// TwinCAT 3 PLC project Anker_Alserbachstrasse
// ProgramVersion: 3.1.4023.0
// libraries:
//   EfficientIO Communicator, * (EfficientIO)
//   Lynus Energy Basic, * (Lynus AG)
//   Lynus Persistent Data V1, * (Lynus AG)
//   Lynus Standards, * (Lynus AG)
//   Tc2_BABasic, * (Beckhoff Automation GmbH)
//   Tc2_Standard, * (Beckhoff Automation GmbH)
//   Tc2_System, * (Beckhoff Automation GmbH)
//   Tc2_Utilities, * (Beckhoff Automation GmbH)
//   Tc3_IotBase, * (Beckhoff Automation GmbH)
//   Tc3_JsonXml, * (Beckhoff Automation GmbH)
//   Tc3_Module, * (Beckhoff Automation GmbH)
// project tree:
//   / FastTask.TcTTO (not stored), MiddleTask.TcTTO, SlowTask.TcTTO (not stored)
//   FBs/ FB_Shelly_Pro1PM.TcPOU, FB_Shelly_Pro1PM_Helper.TcPOU (not stored), FB_TimeSwitch.TcPOU, FB_TimeSwitch_V2.TcPOU
//   POUs/ prg5529Con.TcPOU, prg5529EMS.TcPOU, prgComEffIO.TcPOU, prg5529Grid.TcPOU, prgPersistent.TcPOU, prgRWEffIO.TcPOU, prgVarEffIO.TcPOU (not stored), prg_SystemTime.TcPOU (not stored)
// real-time tasks:
//   TASK FastTask: cycle T#5ms, priority 19, ADS port 350
//   TASK MiddleTask: cycle T#10ms, priority 20, ADS port 351
//   TASK SlowTask: cycle T#20ms, priority 21, ADS port 352
// I/O:
//   DEVICE Device 1 (Beckhoff CCAT)
//   DEVICE Device 2 (CX-BK)
//     Box 1 (CX-BK)
// variable links:
//   Anker_Alserbachstrasse/Anker_Alserbachstrasse Instance <-> Device 2 (CX-BK)/Box 1 (CX-BK)
//     MiddleTask Inputs/prg5529Grid.fbGrid.fbKL3403.byStateCH1 <-> Term 3 (KL3403)/Channel 1/State
//     MiddleTask Inputs/prg5529Grid.fbGrid.fbKL3403.byStateCH2 <-> Term 3 (KL3403)/Channel 2/State
//     MiddleTask Inputs/prg5529Grid.fbGrid.fbKL3403.byStateCH3 <-> Term 3 (KL3403)/Channel 3/State
//     MiddleTask Inputs/prg5529Grid.fbGrid.fbKL3403.iDataInCH1 <-> Term 3 (KL3403)/Channel 1/Data In
//     MiddleTask Inputs/prg5529Grid.fbGrid.fbKL3403.iDataInCH2 <-> Term 3 (KL3403)/Channel 2/Data In
//     MiddleTask Inputs/prg5529Grid.fbGrid.fbKL3403.iDataInCH3 <-> Term 3 (KL3403)/Channel 3/Data In
//     MiddleTask Inputs/prg5529Grid.fbKBusState.uiKBusState_OUT <-> Inputs/State
//     MiddleTask Outputs/prg5529EMS.bQ1Switch <-> Term 2 (KL2408)/Channel 1/Output
//     MiddleTask Outputs/prg5529Grid.fbGrid.fbKL3403.byCntrCH1 <-> Term 3 (KL3403)/Channel 1/Ctrl
//     MiddleTask Outputs/prg5529Grid.fbGrid.fbKL3403.byCntrCH2 <-> Term 3 (KL3403)/Channel 2/Ctrl
//     MiddleTask Outputs/prg5529Grid.fbGrid.fbKL3403.byCntrCH3 <-> Term 3 (KL3403)/Channel 3/Ctrl

CONFIGURATION Anker_Alserbachstrasse
    RESOURCE PLC ON TwinCAT3
        TASK MiddleTask(INTERVAL := T#10ms, PRIORITY := 20);
        PROGRAM prg5529Grid WITH MiddleTask : prg5529Grid;
        PROGRAM prgPersistent WITH MiddleTask : prgPersistent;
        PROGRAM prg5529EMS WITH MiddleTask : prg5529EMS;
        PROGRAM prg5529Con WITH MiddleTask : prg5529Con;
    END_RESOURCE
END_CONFIGURATION

// ---- POUs/prg5529Grid.TcPOU
PROGRAM prg5529Grid
VAR
	fbKBusState		: FB_K_Bus_State;
	fbGrid			: FB_EM_Beckhoff_KL3403;
	lrPowerGrid		: LREAL;							//{#lynus.ag#()}
	lrCounterGrid	: LREAL;							//{#lynus.ag#()}
	lrVoltageGridL1	: LREAL;							//{#lynus.ag#()}
	lrVoltageGridL2	: LREAL;							//{#lynus.ag#()}
	lrVoltageGridL3	: LREAL;							//{#lynus.ag#()}
	uint_BusState	: UINT;								//{#lynus.ag#()}
END_VAR

//The mapping of this function must be linked with the K-Bus State in the E/A Part
fbKBusState(	uiKBusState_OUT=> , 
				b_Kbus_notOk=> , 
				word_ErrorCount=> );
				
//The mapping of this function must be linked with the KL3403 in the E/A Part
fbGrid(
	bEnable:= TRUE, 
	bChannel1Invers:= FALSE,					//Invert power data when transformer are mounted upside down
	bChannel2Invers:= FALSE,
	bChannel3Invers:= FALSE,
	uiCurrentTransformerRatioL1:= 400, 		//Transformer ratio on the secondary side
	uiCurrentTransformerRatioL2:= 400, 
	uiCurrentTransformerRatioL3:= 400, 
	uiKBusState_IN:= fbKBusState.uiKBusState_OUT, 
	stDataEMPower=> , 
	stDataEMCounter=> , 
	stDataEMPowerRealTime=> , 
	stDataEMCounterRealTime=> , 
	diNrOfEM_OUT=> );

lrPowerGrid := fbGrid.stDataEMPower.lrPowerTotal;
	lrCounterGrid := fbGrid.stDataEMCounter.lrTotalCounterEnergy_Consumption;	
		lrVoltageGridL1 := fbGrid.stDataEMPowerRealTime.lrVoltageL1N;
			lrVoltageGridL2 := fbGrid.stDataEMPowerRealTime.lrVoltageL2N;
				lrVoltageGridL3 := fbGrid.stDataEMPowerRealTime.lrVoltageL3N;

				
uint_BusState := fbKbusState.uiKBusState_OUT;

END_PROGRAM

// ---- POUs/prgPersistent.TcPOU
PROGRAM prgPersistent
VAR
	fbUSV		: FB_WritePersistentData_CX81xx;
END_VAR

fbUSV(
	eSaveModeData:= eUSVSaveMode.eSaveWhenPowerfail, 
	bLoadPersistentDataOk=> , 
	bPowerFailDetect=> , 
	bError=> , 
	bySaveProcess=> , 
	dwStorageLast24h=> , 
	udiErrorCode=> );
	
prg_SystemTime();

END_PROGRAM

// ---- POUs/prg5529EMS.TcPOU
PROGRAM prg5529EMS
VAR
	bQ1Switch	AT%Q*	: BOOL;						//{#lynus.ag#()}

	b_Coffee_Manual_On: BOOL;						//{#lynus.ag#()}
	b_Coffee_Manual_Off: BOOL;						//{#lynus.ag#()}
	b_AC_Manual_On: BOOL;							//{#lynus.ag#()}
	b_AC_Manual_Off: BOOL;							//{#lynus.ag#()}
	b_Vitrine_Manual_On: BOOL;						//{#lynus.ag#()}
	b_Vitrine_Manual_Off: BOOL;						//{#lynus.ag#()}
	b_Outside_Manual_On: BOOL;						//{#lynus.ag#()}
	b_Outside_Manual_Off: BOOL;						//{#lynus.ag#()}
	FB_TimeSwitch_Coffee: FB_TimeSwitch_V2;
//	FB_TimeSwitch_Coffee: FB_TimeSwitch;
	FB_TimeSwitch_AC: FB_TimeSwitch_V2;
//	FB_TimeSwitch_AC: FB_TimeSwitch;
	FB_TimeSwitch_Vitrine: FB_TimeSwitch_V2;
//	FB_TimeSwitch_Vitrine: FB_TimeSwitch;
	FB_TimeSwitch_Outside: FB_TimeSwitch_V2;
//	FB_TimeSwitch_Outside: FB_TimeSwitch;
	fbCalcSunriseSunset   		: FB_CalcSunriseSunset;
	todSunrise            		: TOD;
	todSunset             		: TOD;
	fb_GetTimeZoneInfo	:FB_GetTimeZoneInformation;
	b_firstCycle: BOOL;
	RS_Outsidelight: RS;
	r_trig_on: R_trig;
	r_trig_off: R_trig;
	b_Status_CoffeeMaschine: BOOL;					//{#lynus.ag#()}
	// not used any more
	m_error_test	:BOOL;								//{#lynus.ag#()}

END_VAR
VAR PERSISTENT
// opening hours	
	byte_MoFr_Open_Hour		:BYTE;								//{#lynus.ag#()}
	byte_MoFr_Open_Minute	:BYTE;								//{#lynus.ag#()}
	byte_MoFr_Close_Hour	:BYTE;								//{#lynus.ag#()}
	byte_MoFr_Close_Minute	:BYTE;								//{#lynus.ag#()}
	byte_Sa_Open_Hour		:BYTE;								//{#lynus.ag#()}
	byte_Sa_Open_Minute		:BYTE;								//{#lynus.ag#()}
	byte_Sa_Close_Hour		:BYTE;								//{#lynus.ag#()}
	byte_Sa_Close_Minute	:BYTE;								//{#lynus.ag#()}
	byte_So_Open_Hour		:BYTE;								//{#lynus.ag#()}
	byte_So_Open_Minute		:BYTE;								//{#lynus.ag#()}
	byte_So_Close_Hour		:BYTE;								//{#lynus.ag#()}
	byte_So_Close_Minute	:BYTE;								//{#lynus.ag#()}
	
// offset coffeemaschine in hours			
	b_Enable_Control_Coffee		:BOOL;								//{#lynus.ag#()}
	real_Coffee_Offset_Start	:REAL;								//{#lynus.ag#()}
	real_Coffee_Offset_Stop		:REAL;								//{#lynus.ag#()}

// offset AC in hours			
	b_Enable_Control_AC			:BOOL;								//{#lynus.ag#()}
	real_AC_Offset_Start		:REAL;								//{#lynus.ag#()}
	real_AC_Offset_Stop			:REAL;								//{#lynus.ag#()}
	
// offset Vitrine Cooler in hours			
	b_Enable_Control_Vitrine	:BOOL;								//{#lynus.ag#()}
	real_Vitrine_Offset_Start	:REAL;								//{#lynus.ag#()}
	real_Vitrine_Offset_Stop	:REAL;								//{#lynus.ag#()}

// offset outside light in hours			
	b_Enable_Control_Outside	:BOOL;								//{#lynus.ag#()}
	real_Outside_Offset_Start	:REAL;								//{#lynus.ag#()}
	real_Outside_Offset_Stop	:REAL;								//{#lynus.ag#()}
END_VAR

FB_TimeSwitch_Coffee(
	b_Enable:= b_Enable_Control_Coffee, 
	b_StatusOn:= NOT bQ1Switch, 
	structSystemTime:= prg_SystemTime.structSystemTime, 
	byte_MoFr_Open_Hour:= byte_MoFr_Open_Hour , 
	byte_MoFr_Open_Minute:= byte_MoFr_Open_Minute, 
	byte_MoFr_Close_Hour:= byte_MoFr_Close_Hour , 
	byte_MoFr_Close_Minute:= byte_MoFr_Close_Minute, 
	byte_Sa_Open_Hour:= byte_Sa_Open_Hour, 
	byte_Sa_Open_Minute:= byte_Sa_Open_Minute , 
	byte_Sa_Close_Hour:= byte_Sa_Close_Hour , 
	byte_Sa_Close_Minute:= byte_Sa_Close_Minute, 
	byte_So_Open_Hour:= byte_So_Open_Hour, 
	byte_So_Open_Minute:= byte_So_Open_Minute, 
	byte_So_Close_Hour:= byte_So_Close_Hour, 
	byte_So_Close_Minute:= byte_So_Close_Minute, 
	real_Offset_Start:= real_Coffee_Offset_Start , 
	real_Offset_Stop:= real_Coffee_Offset_Stop , 
	b_On_Manual:= b_Coffee_Manual_On, 
	b_Off_Manual:= b_Coffee_Manual_Off, 
	b_Output_On=> , 
	b_Error=> );
	
IF NOT FB_TimeSwitch_Coffee.b_Output_On THEN
	bQ1Switch := TRUE;
ELSIF FB_TimeSwitch_Coffee.b_Output_On THEN
	bQ1Switch := FALSE;
END_IF	
b_Status_CoffeeMaschine := NOT bQ1Switch;
	
FB_TimeSwitch_AC(
	b_Enable:= b_Enable_Control_AC, 
	b_StatusOn:=  prg5529CON.fbShelly[1].bStateP1, 
	structSystemTime:= prg_SystemTime.structSystemTime , 
	byte_MoFr_Open_Hour:= byte_MoFr_Open_Hour , 
	byte_MoFr_Open_Minute:= byte_MoFr_Open_Minute, 
	byte_MoFr_Close_Hour:= byte_MoFr_Close_Hour , 
	byte_MoFr_Close_Minute:= byte_MoFr_Close_Minute, 
	byte_Sa_Open_Hour:= byte_Sa_Open_Hour, 
	byte_Sa_Open_Minute:= byte_Sa_Open_Minute , 
	byte_Sa_Close_Hour:= byte_Sa_Close_Hour , 
	byte_Sa_Close_Minute:= byte_Sa_Close_Minute, 
	byte_So_Open_Hour:= byte_So_Open_Hour, 
	byte_So_Open_Minute:= byte_So_Open_Minute, 
	byte_So_Close_Hour:= byte_So_Close_Hour, 
	byte_So_Close_Minute:= byte_So_Close_Minute, 
	real_Offset_Start:= real_AC_Offset_Start , 
	real_Offset_Stop:= real_AC_Offset_Stop , 
	b_On_Manual:= b_AC_Manual_On, 
	b_Off_Manual:= b_AC_Manual_Off, 
	b_Output_On=> , 
	b_Error=> );

FB_TimeSwitch_Vitrine(
	b_Enable:= b_Enable_Control_Vitrine, 
	b_StatusOn:=  prg5529CON.fbShelly[3].bStateP1, 
	structSystemTime:= prg_SystemTime.structSystemTime , 
	byte_MoFr_Open_Hour:= byte_MoFr_Open_Hour , 
	byte_MoFr_Open_Minute:= byte_MoFr_Open_Minute, 
	byte_MoFr_Close_Hour:= byte_MoFr_Close_Hour , 
	byte_MoFr_Close_Minute:= byte_MoFr_Close_Minute, 
	byte_Sa_Open_Hour:= byte_Sa_Open_Hour, 
	byte_Sa_Open_Minute:= byte_Sa_Open_Minute , 
	byte_Sa_Close_Hour:= byte_Sa_Close_Hour , 
	byte_Sa_Close_Minute:= byte_Sa_Close_Minute, 
	byte_So_Open_Hour:= byte_So_Open_Hour, 
	byte_So_Open_Minute:= byte_So_Open_Minute, 
	byte_So_Close_Hour:= byte_So_Close_Hour, 
	byte_So_Close_Minute:= byte_So_Close_Minute, 
	real_Offset_Start:= real_Vitrine_Offset_Start , 
	real_Offset_Stop:= real_Vitrine_Offset_Stop , 
	b_On_Manual:= b_Vitrine_Manual_On, 
	b_Off_Manual:= b_Vitrine_Manual_Off, 
	b_Output_On=> , 
	b_Error=> );

// Sehlly 5 Outside light
FB_TimeSwitch_Outside(		
	b_Enable:= b_Enable_Control_Outside, 
	b_StatusOn:=  prg5529CON.fbShelly[5].bStateP1 , 
	structSystemTime:= prg_SystemTime.structSystemTime , 
	byte_MoFr_Open_Hour:= byte_MoFr_Open_Hour , 
	byte_MoFr_Open_Minute:= byte_MoFr_Open_Minute, 
	byte_MoFr_Close_Hour:= byte_MoFr_Close_Hour , 
	byte_MoFr_Close_Minute:= byte_MoFr_Close_Minute, 
	byte_Sa_Open_Hour:= byte_Sa_Open_Hour, 
	byte_Sa_Open_Minute:= byte_Sa_Open_Minute , 
	byte_Sa_Close_Hour:= byte_Sa_Close_Hour , 
	byte_Sa_Close_Minute:= byte_Sa_Close_Minute, 
	byte_So_Open_Hour:= byte_So_Open_Hour, 
	byte_So_Open_Minute:= byte_So_Open_Minute, 
	byte_So_Close_Hour:= byte_So_Close_Hour, 
	byte_So_Close_Minute:= byte_So_Close_Minute, 
	real_Offset_Start:= real_Outside_Offset_Start , 
	real_Offset_Stop:= real_Outside_Offset_Stop , 
	b_On_Manual:= b_Outside_Manual_On, 
	b_Off_Manual:= b_Outside_Manual_Off, 
	b_Output_On=> , 
	b_Error=> );
	
// calculate sunset / sunrise
// find out the time details
fb_GetTimeZoneInfo(
	sNetID:= '', 
	bExecute:= prg_SystemTime.structSystemTime.wHour = 4 OR NOT b_firstCycle, 
	tTimeout:= T#5S, 
	bBusy=> , 
	bError=> , 
	nErrID=> , 
	tzID=> , 
	tzInfo=> );
b_firstCycle := TRUE;

fbCalcSunriseSunset(
	fDegreeOfLongitude := 16.3731,   (* Longitude of Vienna *)
	fDegreeOfLatitude := 48.2083,   (* Latitude of Vienna*)
	fReferenceMeridian := SEL( fb_GetTimeZoneInfo.tzID = eTimeZoneID_Daylight ,15,30),  (* Central European Time 15 Winter Timer / 30 Summer Time *)
	dCurrentDate := DT_TO_DATE(SYSTEMTIME_TO_Dt (prg_SystemTime.structSystemTime)),
	todSunrise => todSunrise,
	todSunset => todSunset);
	
r_trig_on (clk := FB_TimeSwitch_Outside.b_Output_On AND DT_TO_TOD(systemtime_to_dt(prg_SystemTime.structSystemTime))< (todSunrise +  T#1H) );
r_trig_off (clk := NOT FB_TimeSwitch_Outside.b_Output_On);

RS_Outsidelight(	Set := r_trig_on.Q OR ((todSunset - T#2H) =  DT_TO_TOD(systemtime_to_dt(prg_SystemTime.structSystemTime)) AND FB_TimeSwitch_Outside.b_Output_On) OR b_Outside_Manual_On ,
					Reset1 := r_trig_off.Q OR ((todSunrise +  T#1H)= DT_TO_TOD(systemtime_to_dt(prg_SystemTime.structSystemTime))) OR b_Outside_Manual_Off,
					Q1 => );

END_PROGRAM

// ---- FBs/FB_TimeSwitch_V2.TcPOU
FUNCTION_BLOCK FB_TimeSwitch_V2
VAR_INPUT
	b_Enable: BOOL;
	b_StatusOn: BOOL;
	structSystemTime: timestruct;
	byte_MoFr_Open_Hour: BYTE;
	byte_MoFr_Open_Minute: BYTE;
	byte_MoFr_Close_Hour: BYTE;
	byte_MoFr_Close_Minute: BYTE;
	byte_Sa_Open_Hour: BYTE;
	byte_Sa_Open_Minute: BYTE;
	byte_Sa_Close_Hour: BYTE;
	byte_Sa_Close_Minute: BYTE;	
	byte_So_Open_Hour: BYTE;
	byte_So_Open_Minute: BYTE;
	byte_So_Close_Hour: BYTE;
	byte_So_Close_Minute: BYTE;
	real_Offset_Start: REAL;
	real_Offset_Stop: REAL;	
	b_On_Manual: BOOL;
	b_Off_Manual: BOOL;
END_VAR
VAR_OUTPUT
	b_Output_On: BOOL;
	b_Error: BOOL;
END_VAR
VAR
	TON_0: ton;
	byte_Day :BYTE;		// 0: Sunday, 1: Monday,....
	time_now             		: TIME;
	time_MoFr_Open             	: TIME;
	time_MoFr_Close             : TIME;
	time_Sa_Open             	: TIME;
	time_Sa_Close             	: TIME;
	time_So_Open             	: TIME;
	time_So_Close             	: TIME;
	

	RS_0: rs;
	R_TRIG_0: r_trig;
	R_TRIG_1: r_trig;
	dt_Test: DATE_AND_TIME;
	tod_test: TIME_OF_DAY;
	time_temp: TIME;
	time_Start_MoFr_Calc: TIME;
	time_Stop_MoFr_Calc: TIME;
	time_Start_Sa_Calc: TIME;
	time_Stop_Sa_Calc: TIME;
	time_Start_So_Calc: TIME;
	time_Stop_So_Calc: TIME;
	
	FB_WeeklyTimeSwitch_MoFr: FB_WeeklyTimeSwitch;
	FB_WeeklyTimeSwitch_Sa: FB_WeeklyTimeSwitch;
	FB_WeeklyTimeSwitch_So: FB_WeeklyTimeSwitch;
	RS_manu: rs;
	b_Auto_on: BOOL;

	R_TRIG_2: r_trig;
	R_TRIG_3: r_trig;
	F_TRIG_0: f_trig;
	R_TRIG_4: r_trig;
	R_TRIG_FirstCycle: r_trig;
	time_Zero             	: TIME;
	
END_VAR
VAR // added by the converter: edge detectors and wires of the graphical bodies
    _w1 : DATE_AND_TIME;
    _w2 : TIME_OF_DAY;
    _w3 : BOOL;
END_VAR

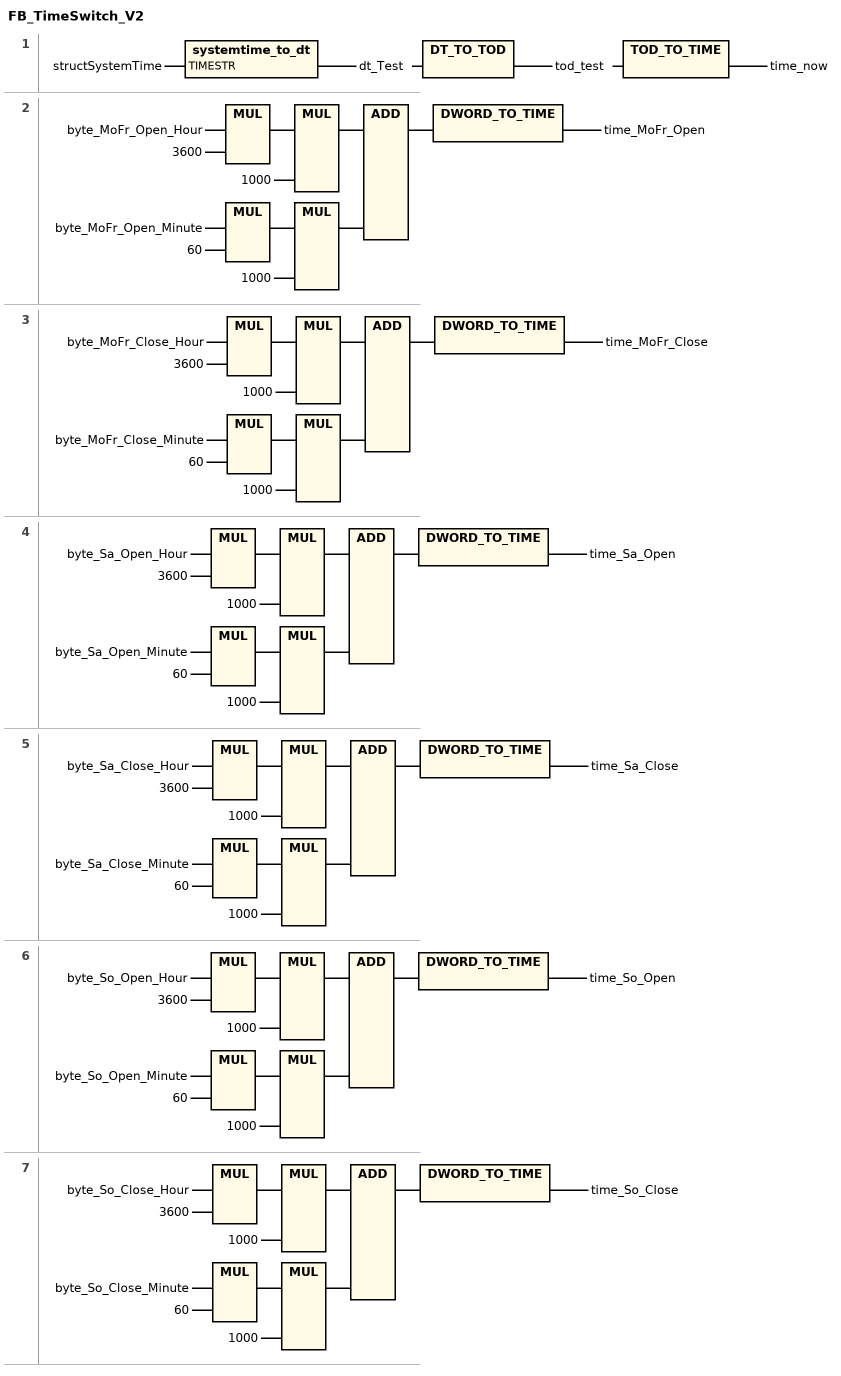
// NETWORK 1
_w1 := systemtime_to_dt(TIMESTR := structSystemTime);
dt_Test := _w1;
_w2 := DT_TO_TOD(_w1);
tod_test := _w2;
time_now := TOD_TO_TIME(_w2);

// NETWORK 2
time_MoFr_Open := DWORD_TO_TIME((byte_MoFr_Open_Hour * 3600) * 1000 + (byte_MoFr_Open_Minute * 60) * 1000);

// NETWORK 3
time_MoFr_Close := DWORD_TO_TIME((byte_MoFr_Close_Hour * 3600) * 1000 + (byte_MoFr_Close_Minute * 60) * 1000);

// NETWORK 4
time_Sa_Open := DWORD_TO_TIME((byte_Sa_Open_Hour * 3600) * 1000 + (byte_Sa_Open_Minute * 60) * 1000);

// NETWORK 5
time_Sa_Close := DWORD_TO_TIME((byte_Sa_Close_Hour * 3600) * 1000 + (byte_Sa_Close_Minute * 60) * 1000);

// NETWORK 6
time_So_Open := DWORD_TO_TIME((byte_So_Open_Hour * 3600) * 1000 + (byte_So_Open_Minute * 60) * 1000);

// NETWORK 7
time_So_Close := DWORD_TO_TIME((byte_So_Close_Hour * 3600) * 1000 + (byte_So_Close_Minute * 60) * 1000);

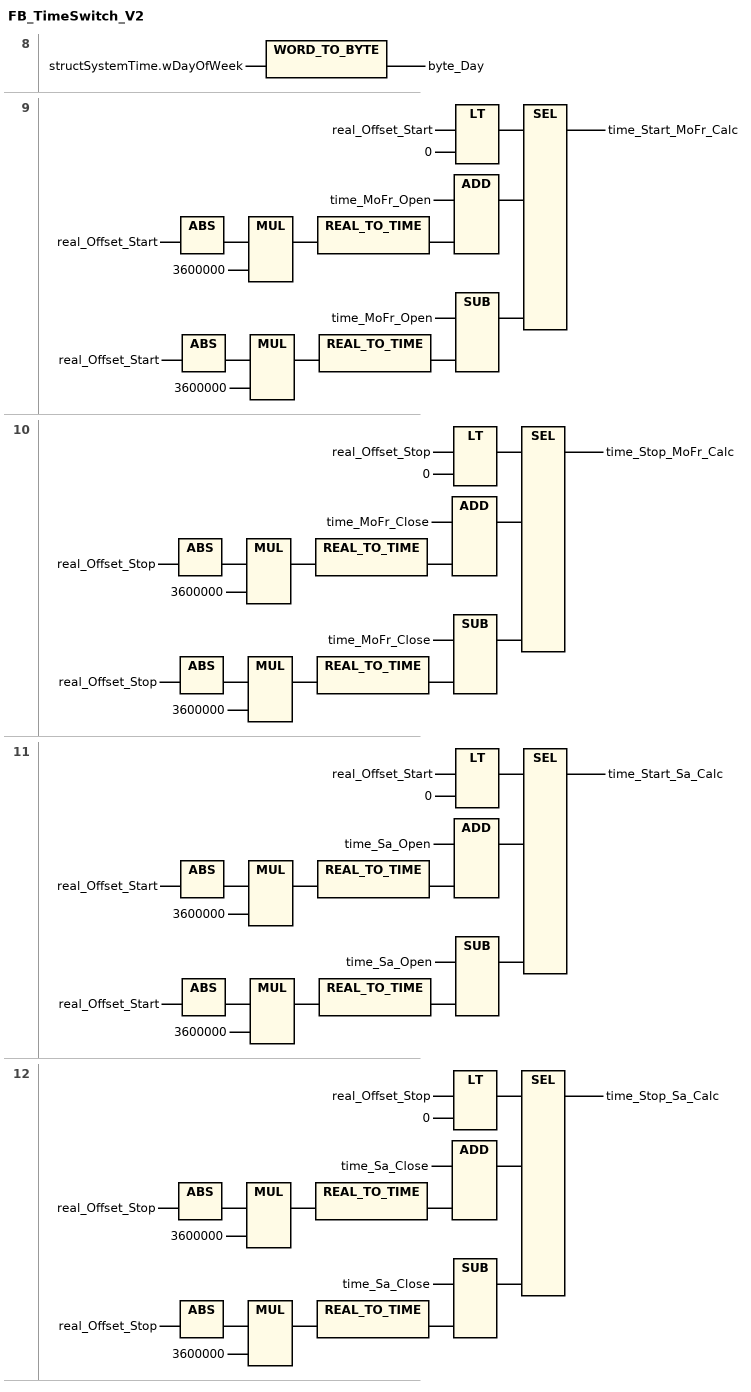
// NETWORK 8
byte_Day := WORD_TO_BYTE(structSystemTime.wDayOfWeek);

// NETWORK 9
time_Start_MoFr_Calc := SEL(real_Offset_Start < 0, time_MoFr_Open + REAL_TO_TIME(ABS(real_Offset_Start) * 3600000), time_MoFr_Open - REAL_TO_TIME(ABS(real_Offset_Start) * 3600000));

// NETWORK 10
time_Stop_MoFr_Calc := SEL(real_Offset_Stop < 0, time_MoFr_Close + REAL_TO_TIME(ABS(real_Offset_Stop) * 3600000), time_MoFr_Close - REAL_TO_TIME(ABS(real_Offset_Stop) * 3600000));

// NETWORK 11
time_Start_Sa_Calc := SEL(real_Offset_Start < 0, time_Sa_Open + REAL_TO_TIME(ABS(real_Offset_Start) * 3600000), time_Sa_Open - REAL_TO_TIME(ABS(real_Offset_Start) * 3600000));

// NETWORK 12
time_Stop_Sa_Calc := SEL(real_Offset_Stop < 0, time_Sa_Close + REAL_TO_TIME(ABS(real_Offset_Stop) * 3600000), time_Sa_Close - REAL_TO_TIME(ABS(real_Offset_Stop) * 3600000));

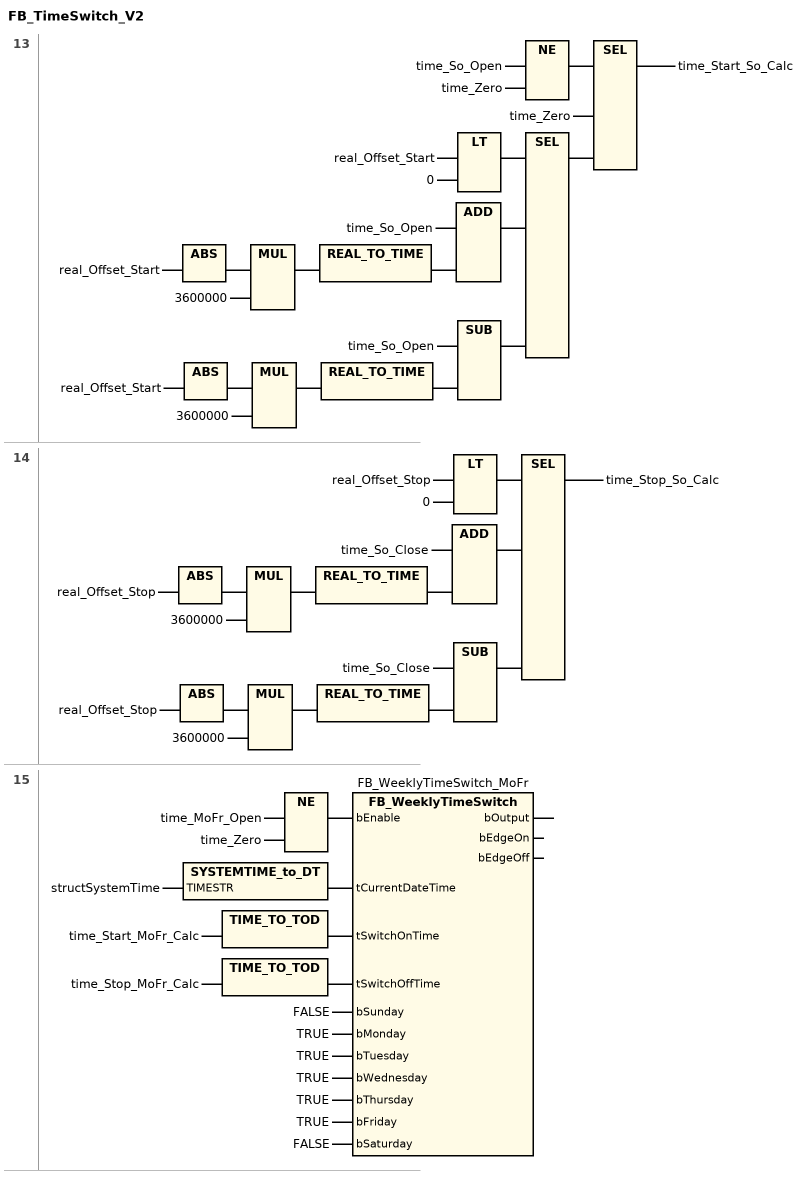
// NETWORK 13
time_Start_So_Calc := SEL(time_So_Open <> time_Zero, time_Zero, SEL(real_Offset_Start < 0, time_So_Open + REAL_TO_TIME(ABS(real_Offset_Start) * 3600000), time_So_Open - REAL_TO_TIME(ABS(real_Offset_Start) * 3600000)));

// NETWORK 14
time_Stop_So_Calc := SEL(real_Offset_Stop < 0, time_So_Close + REAL_TO_TIME(ABS(real_Offset_Stop) * 3600000), time_So_Close - REAL_TO_TIME(ABS(real_Offset_Stop) * 3600000));

// NETWORK 15
FB_WeeklyTimeSwitch_MoFr(
    bEnable := time_MoFr_Open <> time_Zero,
    tCurrentDateTime := SYSTEMTIME_to_DT(TIMESTR := structSystemTime),
    tSwitchOnTime := TIME_TO_TOD(time_Start_MoFr_Calc),
    tSwitchOffTime := TIME_TO_TOD(time_Stop_MoFr_Calc),
    bSunday := FALSE,
    bMonday := TRUE,
    bTuesday := TRUE,
    bWednesday := TRUE,
    bThursday := TRUE,
    bFriday := TRUE,
    bSaturday := FALSE); // FB_WeeklyTimeSwitch

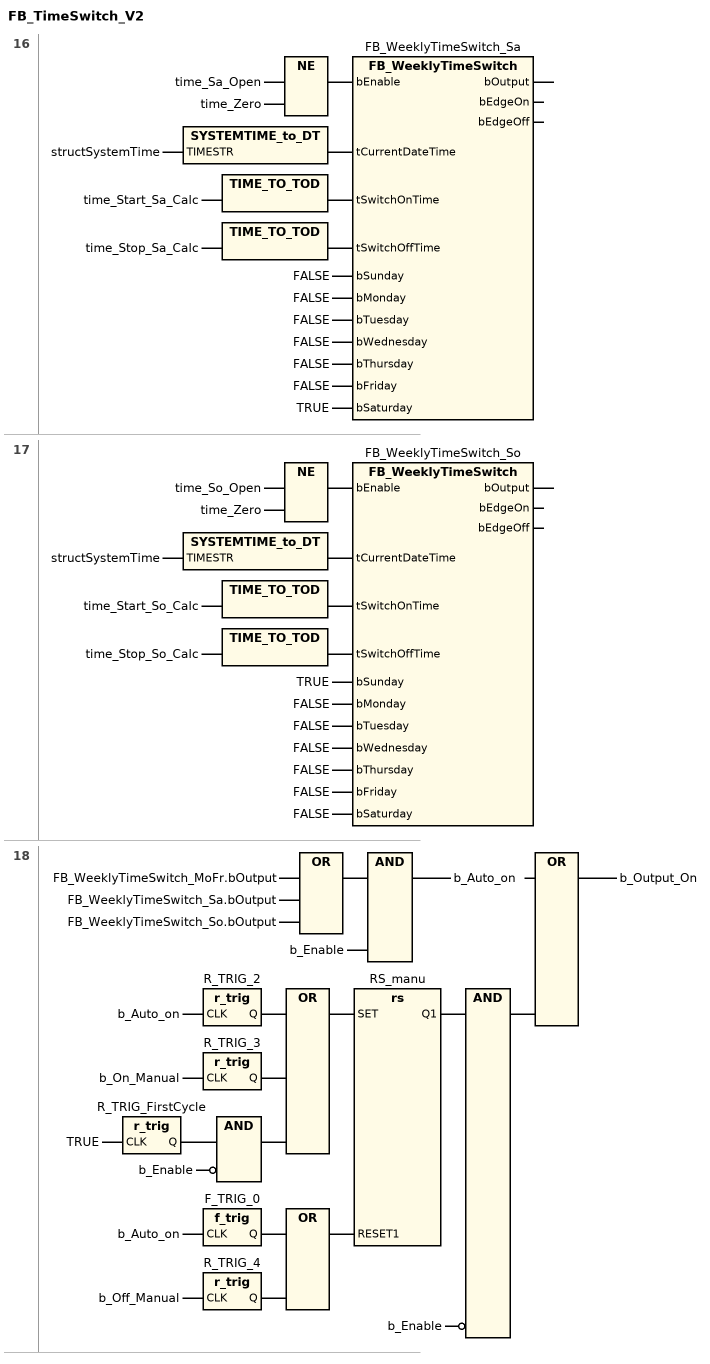
// NETWORK 16
FB_WeeklyTimeSwitch_Sa(
    bEnable := time_Sa_Open <> time_Zero,
    tCurrentDateTime := SYSTEMTIME_to_DT(TIMESTR := structSystemTime),
    tSwitchOnTime := TIME_TO_TOD(time_Start_Sa_Calc),
    tSwitchOffTime := TIME_TO_TOD(time_Stop_Sa_Calc),
    bSunday := FALSE,
    bMonday := FALSE,
    bTuesday := FALSE,
    bWednesday := FALSE,
    bThursday := FALSE,
    bFriday := FALSE,
    bSaturday := TRUE); // FB_WeeklyTimeSwitch

// NETWORK 17
FB_WeeklyTimeSwitch_So(
    bEnable := time_So_Open <> time_Zero,
    tCurrentDateTime := SYSTEMTIME_to_DT(TIMESTR := structSystemTime),
    tSwitchOnTime := TIME_TO_TOD(time_Start_So_Calc),
    tSwitchOffTime := TIME_TO_TOD(time_Stop_So_Calc),
    bSunday := TRUE,
    bMonday := FALSE,
    bTuesday := FALSE,
    bWednesday := FALSE,
    bThursday := FALSE,
    bFriday := FALSE,
    bSaturday := FALSE); // FB_WeeklyTimeSwitch

// NETWORK 18
_w3 := (FB_WeeklyTimeSwitch_MoFr.bOutput OR FB_WeeklyTimeSwitch_Sa.bOutput OR FB_WeeklyTimeSwitch_So.bOutput) AND b_Enable;
b_Auto_on := _w3;
R_TRIG_2(CLK := b_Auto_on); // r_trig
R_TRIG_3(CLK := b_On_Manual); // r_trig
R_TRIG_FirstCycle(CLK := TRUE); // r_trig
F_TRIG_0(CLK := b_Auto_on); // f_trig
R_TRIG_4(CLK := b_Off_Manual); // r_trig
RS_manu(SET := R_TRIG_2.Q OR R_TRIG_3.Q OR R_TRIG_FirstCycle.Q AND NOT b_Enable, RESET1 := F_TRIG_0.Q OR R_TRIG_4.Q); // rs
b_Output_On := _w3 OR RS_manu.Q1 AND NOT b_Enable;

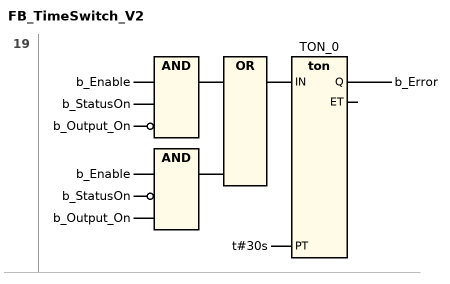
// NETWORK 19
TON_0(IN := b_Enable AND b_StatusOn AND NOT b_Output_On OR b_Enable AND NOT b_StatusOn AND b_Output_On, PT := t#30s); // ton
b_Error := TON_0.Q;

END_FUNCTION_BLOCK

// ---- POUs/prg5529Con.TcPOU
PROGRAM prg5529Con
VAR

	fbShelly				:	ARRAY[1..20] OF FB_Shelly_Pro1PM;
	f_Trig_Busy				:	ARRAY[1..20] OF f_trig;
			
//	fbShelly1				:	FB_Shelly_Pro1PM;
	lrS1P1Power				:	LREAL;			//{#lynus.ag#()}
	lrS1P1Power_kW			:	LREAL;			//{#lynus.ag#()}
	lrS1P1Voltage			:	LREAL;			//{#lynus.ag#()}
	lrS1P1Energy			:	LREAL;			//{#lynus.ag#()}
	lrS1P1Temperature		:	LREAL;			//{#lynus.ag#()}
	bS1P1On					:	BOOL;			//{#lynus.ag#()}
	bS1P1Off				:	BOOL;			//{#lynus.ag#()}
	bS1P1Switch				:	BOOL;			//{#lynus.ag#()}
	
	// Shelly2: 
//	fbShelly2				:	FB_Shelly_Pro1PM;
	lrS2P1Power				:	LREAL;			//{#lynus.ag#()}
	lrS2P1Power_kW			:	LREAL;			//{#lynus.ag#()}
	lrS2P1Voltage			:	LREAL;			//{#lynus.ag#()}
	lrS2P1Energy			:	LREAL;			//{#lynus.ag#()}
	lrS2P1Temperature		:	LREAL;			//{#lynus.ag#()}
	bS2P1On					:	BOOL;			//{#lynus.ag#()}
	bS2P1Off				:	BOOL;			//{#lynus.ag#()}
	bS2P1Switch				:	BOOL;			//{#lynus.ag#()}
	
	// Shelly3: 
//	fbShelly3				:	FB_Shelly_Pro1PM;
	lrS3P1Power				:	LREAL;			//{#lynus.ag#()}
	lrS3P1Power_kW			:	LREAL;			//{#lynus.ag#()}
	lrS3P1Voltage			:	LREAL;			//{#lynus.ag#()}
	lrS3P1Energy			:	LREAL;			//{#lynus.ag#()}
	lrS3P1Temperature		:	LREAL;			//{#lynus.ag#()}
	bS3P1On					:	BOOL;			//{#lynus.ag#()}
	bS3P1Off				:	BOOL;			//{#lynus.ag#()}
	bS3P1Switch				:	BOOL;			//{#lynus.ag#()}
	
	// Shelly4: 
//	fbShelly4				:	FB_Shelly_Pro1PM;
	lrS4P1Power				:	LREAL;			//{#lynus.ag#()}
	lrS4P1Power_kW			:	LREAL;			//{#lynus.ag#()}
	lrS4P1Voltage			:	LREAL;			//{#lynus.ag#()}
	lrS4P1Energy			:	LREAL;			//{#lynus.ag#()}
	lrS4P1Temperature		:	LREAL;			//{#lynus.ag#()}
	bS4P1On					:	BOOL;			//{#lynus.ag#()}
	bS4P1Off				:	BOOL;			//{#lynus.ag#()}
	bS4P1Switch				:	BOOL;			//{#lynus.ag#()}
	
	// Shelly5: 
//	fbShelly5				:	FB_Shelly_Pro1PM;
	lrS5P1Power				:	LREAL;			//{#lynus.ag#()}
	lrS5P1Power_kW			:	LREAL;			//{#lynus.ag#()}
	lrS5P1Voltage			:	LREAL;			//{#lynus.ag#()}
	lrS5P1Energy			:	LREAL;			//{#lynus.ag#()}
	lrS5P1Temperature		:	LREAL;			//{#lynus.ag#()}
	bS5P1On					:	BOOL;			//{#lynus.ag#()}
	bS5P1Off				:	BOOL;			//{#lynus.ag#()}
	bS5P1Switch				:	BOOL;			//{#lynus.ag#()}
	

	// Other
	lrRemainPower_kW		:	LREAL;			//{#lynus.ag#()}
	
	// state maschine for GET requests
	str_Array_IPs			: array[1..30] of STRING(15);			//arrays for IPs
	int_State: INT;													// state
	// Shelly: 


	int_Multiplier_1 			:INT:=1;								// multilpier received values, =2 when external fuse is on, was at the beginning
	int_Multiplier_2 			:INT:=2;								// multilpier received values, =2 when external fuse is on, was at the beginning
	int_Multiplier_3 			:INT:=1;								// multilpier received values, =2 when external fuse is on, was at the beginning
	int_Multiplier_4 			:INT:=2;								// multilpier received values, =2 when external fuse is on, was at the beginning
	int_Multiplier_5 			:INT:=1;								// multilpier received values, =2 when external fuse is on, was at the beginning
	int_TimeoutCounter: ARRAY[1..30] OF INT;	
	int_SuccessCounter: ARRAY[1..30] OF INT;	
	int_ErrorCounter: ARRAY[1..30] OF INT;
	ton_wait: Ton;
	mTest: BOOL;
	m_Error_HTTP: BOOL;							//{#lynus.ag#()}
END_VAR


CASE int_State OF
	0: 		// Init State
	
	// define IPs
	str_Array_IPs[1]	:='10.55.29.131';
	str_Array_IPs[2]	:='10.55.29.132';
	str_Array_IPs[3]	:='10.55.29.133';
	str_Array_IPs[4]	:='10.55.29.134';
	str_Array_IPs[5]	:='10.55.29.135';
	str_Array_IPs[6]	:='';
	str_Array_IPs[7]	:='';
	str_Array_IPs[8]	:='';
	str_Array_IPs[9]	:='';
	str_Array_IPs[10]	:='';
	str_Array_IPs[11]	:='';
	str_Array_IPs[12]	:='';
	str_Array_IPs[13]	:='';
	str_Array_IPs[14]	:='';
	fbShelly[1].sHostname:= str_Array_IPs[1];
	fbShelly[2].sHostname:= str_Array_IPs[2];
	fbShelly[3].sHostname:= str_Array_IPs[3];
	fbShelly[4].sHostname:= str_Array_IPs[4];
	fbShelly[5].sHostname:= str_Array_IPs[5];
 
	
	// =2 for the beginning when bypass fuse is on
	int_Multiplier_1:=1;
	int_Multiplier_2:=2;
	int_Multiplier_3:=1;
	int_Multiplier_4:=2;
	int_Multiplier_5:=1;
	
	IF str_Array_IPs[1] <> '' THEN
		int_State :=1;
	END_IF
		
	1: 		// request
	
		fbShelly[int_State].bStart:= TRUE;
		fbShelly[int_State].bOnP1:= bS1P1On;
		fbShelly[int_State].bOffP1:= bS1P1Off;
	
		f_Trig_Busy[int_State](CLK :=fbShelly[int_State].bBusy);
			
		// go to next state
		IF f_Trig_Busy[int_State].Q  AND NOT fbShelly[int_State].bError THEN	
			int_SuccessCounter[int_State]	:= int_SuccessCounter[int_State]+1;
			lrS1P1Power 	:= 	fbShelly[int_State].lrpowerP1 * int_Multiplier_1;
			lrS1P1Energy 	:= 	fbShelly[int_State].lrenergyP1 * int_Multiplier_1;
			lrS1P1Voltage	:=	fbShelly[int_State].lrvoltageP1; 
			lrS1P1Temperature :=fbShelly[int_State].lrTemperatureP1;
			bS1P1Switch		:=	fbShelly[int_State].bStateP1;
		ELSIF  f_Trig_Busy[int_State].Q  AND fbShelly[int_State].bError THEN
			int_ErrorCounter[int_State]	:= int_ErrorCounter[int_State]+1;
		END_IF
		IF 	int_state < 20 AND str_Array_IPs[int_State+1] <> '' AND f_Trig_Busy[int_State].Q  THEN	
			fbShelly[int_State].bStart		:= FALSE;
			int_State := int_State+1;
		ELSIF  (str_Array_IPs[int_State+1] = '' OR int_state > 20) AND f_Trig_Busy[int_State].Q THEN
			fbShelly[int_State].bStart		:= FALSE;
			int_State := 100;			// wait state for new run
		END_IF		
	
	2: 		// request
	
		fbShelly[int_State].bStart:= TRUE;
		fbShelly[int_State].bOnP1:= bS2P1On;
		fbShelly[int_State].bOffP1:= bS2P1Off;
	
		f_Trig_Busy[int_State](CLK :=fbShelly[int_State].bBusy);
			
		// go to next state
		IF f_Trig_Busy[int_State].Q  AND NOT fbShelly[int_State].bError THEN	
			int_SuccessCounter[int_State]	:= int_SuccessCounter[int_State]+1;
			lrS2P1Power 	:= 	fbShelly[int_State].lrpowerP1 * int_Multiplier_2;
			lrS2P1Energy 	:= 	fbShelly[int_State].lrenergyP1 * int_Multiplier_2;
			lrS2P1Temperature :=fbShelly[int_State].lrTemperatureP1;
			lrS2P1Voltage	:=	fbShelly[int_State].lrvoltageP1; 
			bS2P1Switch		:=	fbShelly[int_State].bStateP1;
		ELSIF  f_Trig_Busy[int_State].Q  AND fbShelly[int_State].bError THEN
			int_ErrorCounter[int_State]	:= int_ErrorCounter[int_State]+1;
		END_IF
		IF 	int_state < 20 AND str_Array_IPs[int_State+1] <> '' AND f_Trig_Busy[int_State].Q  THEN	
			fbShelly[int_State].bStart		:= FALSE;
			int_State := int_State+1;
		ELSIF  (str_Array_IPs[int_State+1] = '' OR int_state > 20) AND f_Trig_Busy[int_State].Q THEN
			fbShelly[int_State].bStart		:= FALSE;
			int_State := 100;			// wait state for new run
		END_IF	
		
	3: 		// request
		fbShelly[int_State].bStart:= TRUE;
		fbShelly[int_State].bOnP1:= bS3P1On;
		fbShelly[int_State].bOffP1:= bS3P1Off;
	
		f_Trig_Busy[int_State](CLK :=fbShelly[int_State].bBusy);
			
		// go to next state
		IF f_Trig_Busy[int_State].Q  AND NOT fbShelly[int_State].bError THEN	
			int_SuccessCounter[int_State]	:= int_SuccessCounter[int_State]+1;
			lrS3P1Power 	:= 	fbShelly[int_State].lrpowerP1 * int_Multiplier_3;
			lrS3P1Energy 	:= 	fbShelly[int_State].lrenergyP1 * int_Multiplier_3;
			lrS3P1Temperature :=fbShelly[int_State].lrTemperatureP1;
			lrS3P1Voltage	:=	fbShelly[int_State].lrvoltageP1; 
			bS3P1Switch		:=	fbShelly[int_State].bStateP1;
		ELSIF  f_Trig_Busy[int_State].Q  AND fbShelly[int_State].bError THEN
			int_ErrorCounter[int_State]	:= int_ErrorCounter[int_State]+1;
		END_IF
		IF 	int_state < 20 AND str_Array_IPs[int_State+1] <> '' AND f_Trig_Busy[int_State].Q  THEN	
			fbShelly[int_State].bStart		:= FALSE;
			int_State := int_State+1;
		ELSIF  (str_Array_IPs[int_State+1] = '' OR int_state > 20) AND f_Trig_Busy[int_State].Q THEN
			fbShelly[int_State].bStart		:= FALSE;
			int_State := 100;			// wait state for new run
		END_IF	
	4: 		// request
	
		fbShelly[int_State].bStart:= TRUE;
		fbShelly[int_State].bOnP1:= bS4P1On;
		fbShelly[int_State].bOffP1:= bS4P1Off;
	
		f_Trig_Busy[int_State](CLK :=fbShelly[int_State].bBusy);
			
		// go to next state
		IF f_Trig_Busy[int_State].Q  AND NOT fbShelly[int_State].bError THEN	
			int_SuccessCounter[int_State]	:= int_SuccessCounter[int_State]+1;
			lrS4P1Power 	:= 	fbShelly[int_State].lrpowerP1 * int_Multiplier_4;
			lrS4P1Energy 	:= 	fbShelly[int_State].lrenergyP1 * int_Multiplier_4;
			lrS4P1Temperature :=fbShelly[int_State].lrTemperatureP1;
			lrS4P1Voltage	:=	fbShelly[int_State].lrvoltageP1; 
			bS4P1Switch		:=	fbShelly[int_State].bStateP1;
		ELSIF  f_Trig_Busy[int_State].Q  AND fbShelly[int_State].bError THEN
			int_ErrorCounter[int_State]	:= int_ErrorCounter[int_State]+1;
		END_IF
		IF 	int_state < 20 AND str_Array_IPs[int_State+1] <> '' AND f_Trig_Busy[int_State].Q  THEN	
			fbShelly[int_State].bStart		:= FALSE;
			int_State := int_State+1;
		ELSIF  (str_Array_IPs[int_State+1] = '' OR int_state > 20) AND f_Trig_Busy[int_State].Q THEN
			fbShelly[int_State].bStart		:= FALSE;
			int_State := 100;			// wait state for new run
		END_IF
		
	5: 		// request
	
		fbShelly[int_State].bStart:= TRUE;
		fbShelly[int_State].bOnP1:= bS5P1On;
		fbShelly[int_State].bOffP1:= bS5P1Off;
	
		f_Trig_Busy[int_State](CLK :=fbShelly[int_State].bBusy);
			
		// go to next state
		IF f_Trig_Busy[int_State].Q  AND NOT fbShelly[int_State].bError THEN	
			int_SuccessCounter[int_State]	:= int_SuccessCounter[int_State]+1;
			lrS5P1Power 	:= 	fbShelly[int_State].lrpowerP1 * int_Multiplier_5;
			lrS5P1Energy 	:= 	fbShelly[int_State].lrenergyP1 * int_Multiplier_5;
			lrS5P1Temperature :=fbShelly[int_State].lrTemperatureP1;
			lrS5P1Voltage	:=	fbShelly[int_State].lrvoltageP1; 
			bS5P1Switch		:=	fbShelly[int_State].bStateP1;
		ELSIF  f_Trig_Busy[int_State].Q  AND fbShelly[int_State].bError THEN
			int_ErrorCounter[int_State]	:= int_ErrorCounter[int_State]+1;
		END_IF
		IF 	int_state < 20 AND str_Array_IPs[int_State+1] <> '' AND f_Trig_Busy[int_State].Q  THEN	
			fbShelly[int_State].bStart		:= FALSE;
			int_State := int_State+1;
		ELSIF  (str_Array_IPs[int_State+1] = '' OR int_state > 20) AND f_Trig_Busy[int_State].Q THEN
			fbShelly[int_State].bStart		:= FALSE;
			int_State := 100;			// wait state for new run
		END_IF	
	
	100:		// wait state
	ton_wait.IN :=TRUE;
	IF ton_wait.Q THEN
		ton_wait.IN :=FALSE;
		int_State := 1;
	END_IF	
END_CASE


// Shelly communication

fbShelly[1](tDelayRequest:= T#0S, );
fbShelly[2](tDelayRequest:= T#0S, );
fbShelly[3](tDelayRequest:= T#0S, );
fbShelly[4](tDelayRequest:= T#0S, );
fbShelly[5](tDelayRequest:= T#0S, );


// wait
ton_wait(PT:=T#3S);


	
// re-calc to kW
lrS1P1Power_kW := lrS1P1Power / 1000;
lrS2P1Power_kW := lrS2P1Power / 1000;
lrS3P1Power_kW := lrS3P1Power / 1000;
lrS4P1Power_kW := lrS4P1Power / 1000;
lrS5P1Power_kW := lrS5P1Power / 1000;
				
// Other
lrRemainPower_kW := LIMIT(0, prg5529Grid.lrPowerGrid - (lrS1P1Power_kW + lrS2P1Power_kW + lrS3P1Power_kW + lrS4P1Power_kW + lrS5P1Power_kW), 999999);
	
	
// on / off commands from EMS
// Klima Shelly 1
fbShelly[1].bEnableControl := TRUE; 	// prg5529EMS.FB_TimeSwitch_AC.b_Enable;
IF prg5529EMS.FB_TimeSwitch_AC.b_Output_On AND NOT fbShelly[1].bStateP1 THEN
	bS1P1On :=TRUE;
ELSE
	bS1P1On := FALSE;
END_IF
IF NOT prg5529EMS.FB_TimeSwitch_AC.b_Output_On AND fbShelly[1].bStateP1 THEN
	bS1P1Off :=TRUE;
ELSE
	bS1P1Off := FALSE;
END_IF
// Kühlvitrine Shelly 3
fbShelly[3].bEnableControl := TRUE; 	// prg5529EMS.FB_TimeSwitch_Vitrine.b_Enable;
IF prg5529EMS.FB_TimeSwitch_Vitrine.b_Output_On AND NOT fbShelly[3].bStateP1 THEN
	bS3P1On :=TRUE;
ELSE
	bS3P1On := FALSE;
END_IF
IF NOT prg5529EMS.FB_TimeSwitch_Vitrine.b_Output_On AND fbShelly[3].bStateP1 THEN
	bS3P1Off :=TRUE;
ELSE
	bS3P1Off := FALSE;
END_IF


// Außenbeleuchtung Shelly 5
fbShelly[5].bEnableControl := TRUE; 	// prg5529EMS.FB_TimeSwitch_Outside.b_Enable;
IF prg5529EMS.RS_Outsidelight.Q1 AND NOT fbShelly[5].bStateP1 THEN
	bS5P1On :=TRUE;
ELSE
	bS5P1On := FALSE;
END_IF
IF NOT prg5529EMS.RS_Outsidelight.Q1 AND fbShelly[5].bStateP1 THEN
	bS5P1Off :=TRUE;
ELSE
	bS5P1Off := FALSE;
END_IF


// error bit to cloud 

m_Error_HTTP := fbShelly[1].bError OR fbShelly[3].bError OR fbShelly[5].bError;

END_PROGRAM

// ---- FBs/FB_Shelly_Pro1PM.TcPOU
FUNCTION_BLOCK FB_Shelly_Pro1PM
VAR_INPUT
	bStart				: BOOL;
	tDelayRequest		: TIME;				//Timer for delay before start with the next read or write Request
	sHostname			: STRING(255);		//Hostname or IP Adress from the Server
	bOnP1				: BOOL;
	bOffP1				: BOOL;
	bEnableControl		: BOOL;
END_VAR

VAR_OUTPUT
	bValidResult				: BOOL;															//Valid Result received from Server
    bBusy						: BOOL;															//Function is Busy
    bError						: BOOL;															//Error sucess
	bDone						: BOOL;															//True after the decoding from the received Json File
	bConnected					: BOOL;															//Connection to the Server
	hrErrorCode       			: HRESULT;														//Error Result from Http Client
	lrpowerP1					: LREAL;														//Received Value
	lrvoltageP1					: LREAL;														//Received Value
	lrenergyP1					: LREAL;														//Received Value
	lrTemperatureP1				: LREAL;														//Received Value
	bStateP1					: BOOL;
END_VAR

VAR
	fbClient					: FB_IotHttpClient;
	fbHttpGet					: FB_Shelly_Pro1PM_Helper;
	timStartRequest				: TON;															//Timer to Start the Request
	FPStartRequest				: R_TRIG;														//Internal positive Edge
	FPDone						: R_TRIG;														//Internal positive Edge
	FNStart						: F_TRIG;														//Internal negative Edge
	SwitchOnP1					: R_TRIG;
	SwitchOffP1					: R_TRIG;
	rs_Switch_ON: Rs;
	rs_Switch_OFF: RS;
	x: INT;
END_VAR

bError := FALSE;
(*------------------------------------------------------------------------------------Configure HTTP Client------------------------------------------------------------------------------------------------------*)

fbClient.sHostName := sHostname;
fbClient.tConnectionTimeout := T#25S;

IF NOT fbClient.bConfigured THEN 
	fbClient.nHostPort:= 80;
	fbClient.bKeepAlive := TRUE;
	fbClient.tConnectionTimeout := T#25S;
END_IF


//Timer to start the Request
FPStartRequest(CLK:= bStart, Q=> );
timStartRequest(	IN:= fbClient.bConfigured AND bStart AND NOT timStartRequest.Q, 
					PT:= tDelayRequest, 
					Q=> , 
					ET=> );
IF ((timStartRequest.Q AND NOT bBusy) OR (FPStartRequest.Q AND NOT bBusy AND fbClient.bConfigured)) THEN 
	fbHttpGet.bSend := TRUE; 
	x:=x+1;
END_IF

				
//Http Get Function
fbHttpGet(
	lrapowerP1 => lrpowerP1, 
	lrvoltageP1 => lrvoltageP1, 
	lraenergyP1 => lrenergyP1,
	lrTemperatureP1 => lrTemperatureP1,
	bSend:= , 
	fbClient:= fbClient, 
	bBusy=> bBusy, 
	bError=> ,
	sContentS0=> ,
	bStateP1=>bStateP1 );


fbHttpGet.bSend := FALSE;

FPDone(CLK:= bDone, Q=> );

// zum testen ob dadurch die verbindung aufrechtbleibt nach dem schalten 
// --> error geht nicht mehr low!
// IF NOT bError  THEN
	fbClient.Execute();
// ELSE
//	fbClient.Disconnect();
// END_IF

//Error
IF fbHttpGet.bError OR fbClient.bError THEN bError := TRUE; ELSE bError := FALSE; END_IF	
	hrErrorCode := fbClient.hrErrorCode;
	

// Relay Control, Switch P1
SwitchOnP1(CLK:=bOnP1);
rs_Switch_ON(	Set:= SwitchOnP1.Q AND bEnableControl,
				Reset1 := bStateP1);	// OR fbHttpGet.timTimeoutSwitch.Q);
				
IF rs_Switch_ON.Q1 AND bEnableControl THEN
	fbHttpGet.bSetOnP1 := TRUE;
ELSE
	fbHttpGet.bSetOnP1 := FALSE;
END_IF

SwitchOffP1(CLK:=bOffP1);
rs_Switch_OFF(	Set:= SwitchOffP1.Q AND bEnableControl,
				Reset1 := NOT bStateP1);	// OR fbHttpGet.timTimeoutSwitch.Q);
				
IF rs_Switch_OFF.Q1 AND bEnableControl THEN
	fbHttpGet.bSetOffP1 := TRUE;
ELSE
	fbHttpGet.bSetOffP1 := FALSE;
END_IF

END_FUNCTION_BLOCK

// ---- FBs/FB_TimeSwitch.TcPOU
FUNCTION_BLOCK FB_TimeSwitch
VAR_INPUT
	b_Enable: BOOL;
	b_StatusOn: BOOL;
	structSystemTime: timestruct;
	byte_MoFr_Open_Hour: BYTE;
	byte_MoFr_Open_Minute: BYTE;
	byte_MoFr_Close_Hour: BYTE;
	byte_MoFr_Close_Minute: BYTE;
	byte_Sa_Open_Hour: BYTE;
	byte_Sa_Open_Minute: BYTE;
	byte_Sa_Close_Hour: BYTE;
	byte_Sa_Close_Minute: BYTE;	
	byte_So_Open_Hour: BYTE;
	byte_So_Open_Minute: BYTE;
	byte_So_Close_Hour: BYTE;
	byte_So_Close_Minute: BYTE;
	real_Offset_Start: REAL;
	real_Offset_Stop: REAL;	
	b_On_Manual: BOOL;
	b_Off_Manual: BOOL;
END_VAR
VAR_OUTPUT
	b_Output_On: BOOL;
	b_Error: BOOL;
END_VAR
VAR
	TON_0: ton;
	byte_Day :BYTE;		// 0: Sunday, 1: Monday,....
	time_now             		: TIME;
	time_MoFr_Open             	: TIME;
	time_MoFr_Close             : TIME;
	time_Sa_Open             	: TIME;
	time_Sa_Close             	: TIME;
	time_So_Open             	: TIME;
	time_So_Close             	: TIME;
	

	RS_0: rs;
	R_TRIG_0: r_trig;
	R_TRIG_1: r_trig;
	dt_Test: DATE_AND_TIME;
	tod_test: TIME_OF_DAY;
	time_temp: TIME;
	time_Start_MoFr_Calc: TIME;
	time_Stop_MoFr_Calc: TIME;
	time_Start_Sa_Calc: TIME;
	time_Stop_Sa_Calc: TIME;
	time_Start_So_Calc: TIME;
	time_Stop_So_Calc: TIME;
	
END_VAR
VAR // added by the converter: edge detectors and wires of the graphical bodies
    _w1 : DATE_AND_TIME;
    _w2 : TIME_OF_DAY;
END_VAR

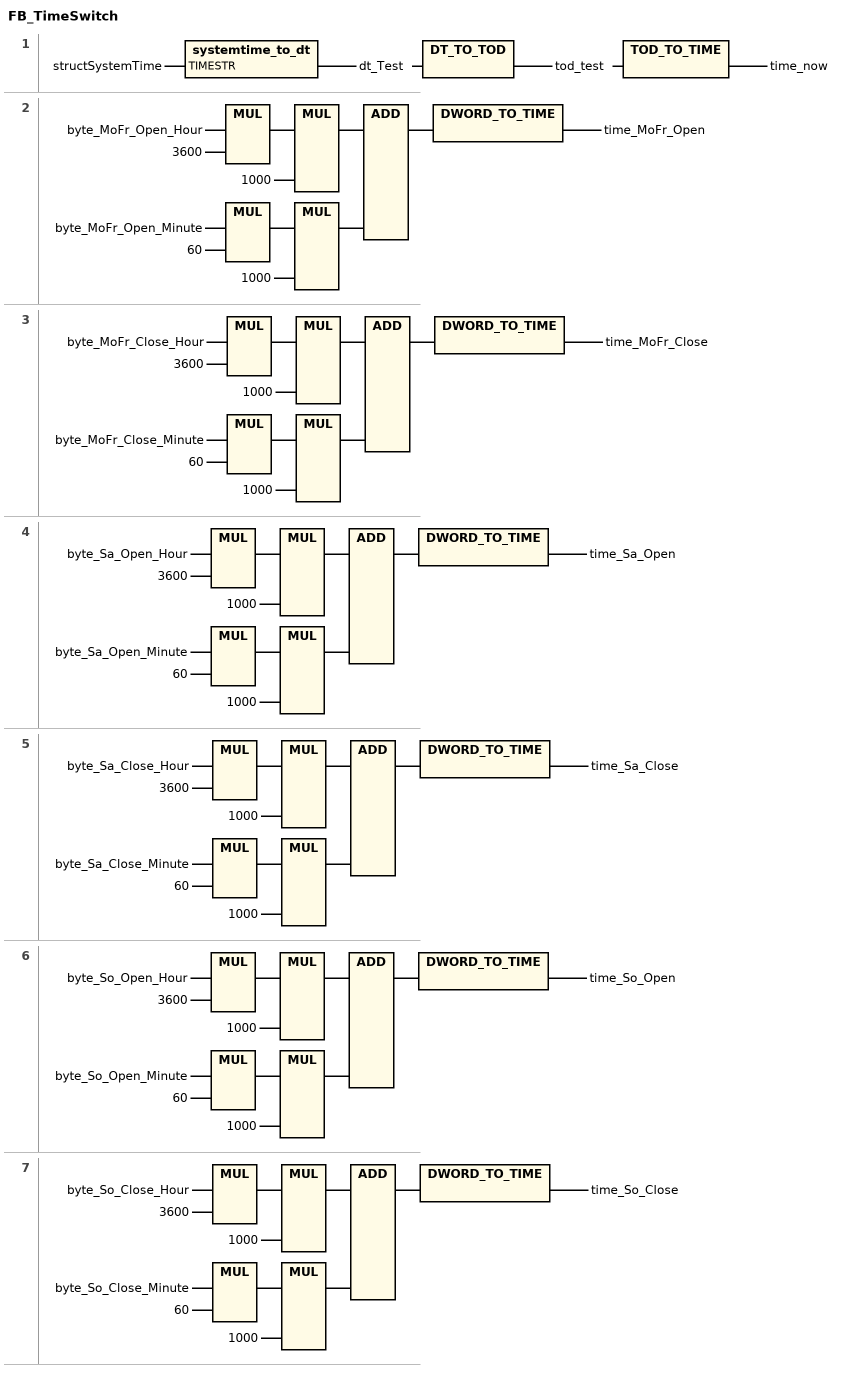
// NETWORK 1
_w1 := systemtime_to_dt(TIMESTR := structSystemTime);
dt_Test := _w1;
_w2 := DT_TO_TOD(_w1);
tod_test := _w2;
time_now := TOD_TO_TIME(_w2);

// NETWORK 2
time_MoFr_Open := DWORD_TO_TIME((byte_MoFr_Open_Hour * 3600) * 1000 + (byte_MoFr_Open_Minute * 60) * 1000);

// NETWORK 3
time_MoFr_Close := DWORD_TO_TIME((byte_MoFr_Close_Hour * 3600) * 1000 + (byte_MoFr_Close_Minute * 60) * 1000);

// NETWORK 4
time_Sa_Open := DWORD_TO_TIME((byte_Sa_Open_Hour * 3600) * 1000 + (byte_Sa_Open_Minute * 60) * 1000);

// NETWORK 5
time_Sa_Close := DWORD_TO_TIME((byte_Sa_Close_Hour * 3600) * 1000 + (byte_Sa_Close_Minute * 60) * 1000);

// NETWORK 6
time_So_Open := DWORD_TO_TIME((byte_So_Open_Hour * 3600) * 1000 + (byte_So_Open_Minute * 60) * 1000);

// NETWORK 7
time_So_Close := DWORD_TO_TIME((byte_So_Close_Hour * 3600) * 1000 + (byte_So_Close_Minute * 60) * 1000);

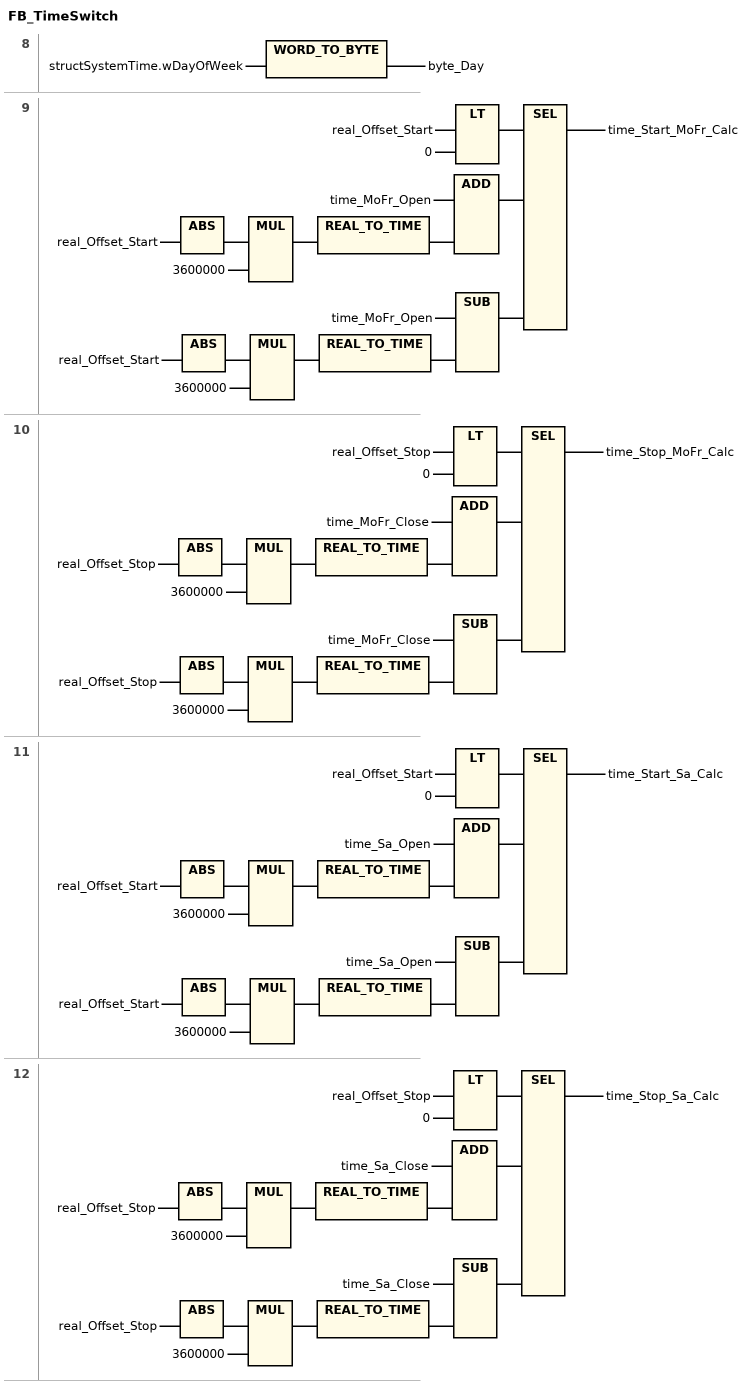
// NETWORK 8
byte_Day := WORD_TO_BYTE(structSystemTime.wDayOfWeek);

// NETWORK 9
time_Start_MoFr_Calc := SEL(real_Offset_Start < 0, time_MoFr_Open + REAL_TO_TIME(ABS(real_Offset_Start) * 3600000), time_MoFr_Open - REAL_TO_TIME(ABS(real_Offset_Start) * 3600000));

// NETWORK 10
time_Stop_MoFr_Calc := SEL(real_Offset_Stop < 0, time_MoFr_Close + REAL_TO_TIME(ABS(real_Offset_Stop) * 3600000), time_MoFr_Close - REAL_TO_TIME(ABS(real_Offset_Stop) * 3600000));

// NETWORK 11
time_Start_Sa_Calc := SEL(real_Offset_Start < 0, time_Sa_Open + REAL_TO_TIME(ABS(real_Offset_Start) * 3600000), time_Sa_Open - REAL_TO_TIME(ABS(real_Offset_Start) * 3600000));

// NETWORK 12
time_Stop_Sa_Calc := SEL(real_Offset_Stop < 0, time_Sa_Close + REAL_TO_TIME(ABS(real_Offset_Stop) * 3600000), time_Sa_Close - REAL_TO_TIME(ABS(real_Offset_Stop) * 3600000));

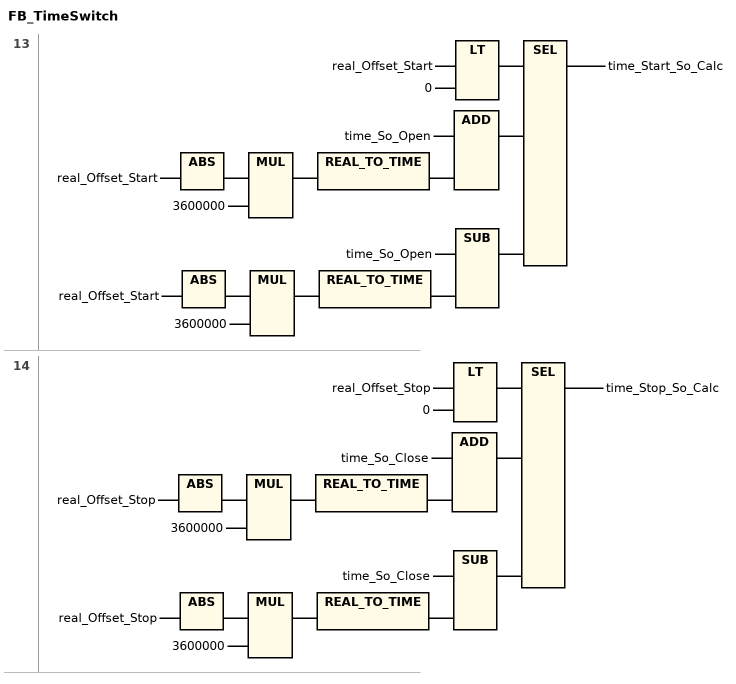
// NETWORK 13
time_Start_So_Calc := SEL(real_Offset_Start < 0, time_So_Open + REAL_TO_TIME(ABS(real_Offset_Start) * 3600000), time_So_Open - REAL_TO_TIME(ABS(real_Offset_Start) * 3600000));

// NETWORK 14
time_Stop_So_Calc := SEL(real_Offset_Stop < 0, time_So_Close + REAL_TO_TIME(ABS(real_Offset_Stop) * 3600000), time_So_Close - REAL_TO_TIME(ABS(real_Offset_Stop) * 3600000));

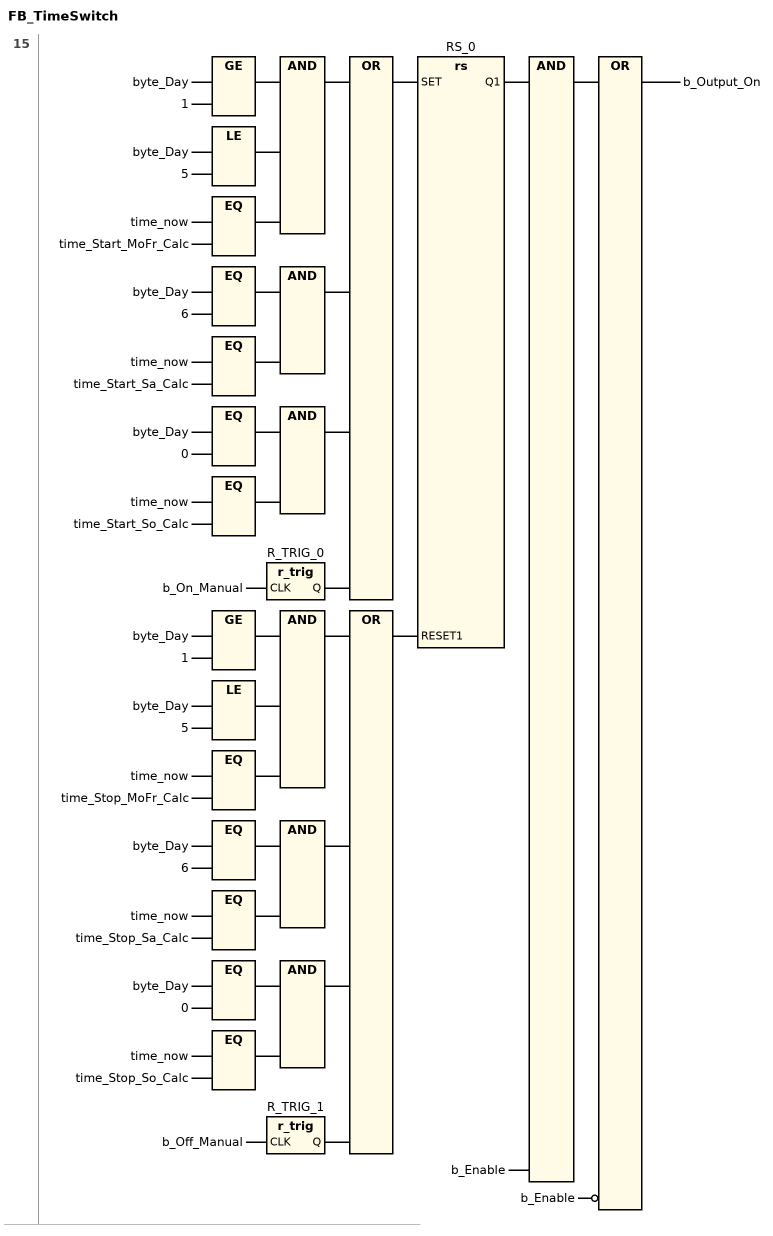
// NETWORK 15
R_TRIG_0(CLK := b_On_Manual); // r_trig
R_TRIG_1(CLK := b_Off_Manual); // r_trig
RS_0(SET := byte_Day >= 1 AND byte_Day <= 5 AND time_now = time_Start_MoFr_Calc OR byte_Day = 6 AND time_now = time_Start_Sa_Calc OR byte_Day = 0 AND time_now = time_Start_So_Calc OR R_TRIG_0.Q, RESET1 := byte_Day >= 1 AND byte_Day <= 5 AND time_now = time_Stop_MoFr_Calc OR byte_Day = 6 AND time_now = time_Stop_Sa_Calc OR byte_Day = 0 AND time_now = time_Stop_So_Calc OR R_TRIG_1.Q); // rs
b_Output_On := RS_0.Q1 AND b_Enable OR NOT b_Enable;

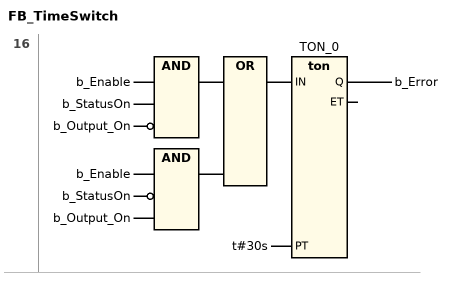
// NETWORK 16
TON_0(IN := b_Enable AND b_StatusOn AND NOT b_Output_On OR b_Enable AND NOT b_StatusOn AND b_Output_On, PT := t#30s); // ton
b_Error := TON_0.Q;

END_FUNCTION_BLOCK

// ---- POUs/prgComEffIO.TcPOU
PROGRAM prgComEffIO
VAR
	fbCom		: FB_MqttCommunicator;
END_VAR

fbCom(
	bConnect:= TRUE, 
	sUserName:= 'd7aecbab-7f4e-4acb-b33b-24861f013074', 
	sUserPassword:= '3abb15af-0787-45ea-b3af-d708d75008a0', 
	eSavePositionCertificate:= eSavePositionOnPLC.ePostionHardDisk, 
	bConnected=> , 
	bError=> , 
	hrErrorCode=> , 
	eConnectionState=> , 
	eErrorMessage_Out=> );

END_PROGRAM

// ---- POUs/prgRWEffIO.TcPOU
PROGRAM prgRWEffIO
VAR
	fbRW1		: FB_ReadWrite_V2;
END_VAR

fbRW1(
	eUploadType:= 3, // Change + 5 min Intervall 
	bBusy=> , 
	bError=> , 
	udiErrorCodeOut=> , 
	eErrorReadWrite_Out=> );

END_PROGRAM
